TYPE ST_3024_ReturnToRoute EXTENDS ST_SupervisorHeader :
	STRUCT
	END_STRUCT
END_TYPE

(* stored: Version 1.1.0.1
   DUT ST_3024_ReturnToRoute: Id {fdadc0c3-0fac-49a0-8d12-66b962a221c1} *)
